TYPE ST_HW_OutputsEtherCAT_Bridge :
(**************************************************************************************
 * 	Application		:	BoxControl Framework
 *	Revision		:	$Revision: 355211 $
 *	Revision date	:	$Date: 2015-09-22 11:14:21 +0200 (Tue, 22 Sep 2015) $
 *	Last changed by	:	$Author: b7bolm $
 *	URL				:	$URL: http://almscdc.swisslog.com/repo/SWPD/Development/BoxControlFramework/20_Release/trunk/01_Software/BoxControlFramework/BoxControlFramework/JumpStart/11_Library/10_Application/11_Communication/12_MFCS/11_SIS/10_Base/FB_SIS_BaseDriver.TcPOU $
 *
 *	Purpose			:	Data for conveyor Subsystem interface over EtherCAT
 *
 * ------------------------------------------------------------------------------------
 *	Copyright Swisslog [IP AG], Switzerland. All rights reserved.
 * 
 * ------------------------------------------------------------------------------------
 *	
 * 	Revision History: 
 *
 * 	VERSION			DATE			INITIALS			DESCRIPTION
 *	0.1				01.01.2001		swl					Example
 *
 **************************************************************************************)
STRUCT
	STI					: ARRAY[1..20] OF ST_HW_InOutputsSTI_EtherCAT_Conveyor; // STI interface
END_STRUCT
END_TYPE

(* stored: Version 1.1.0.1, ProductVersion 3.1.4022.12
   DUT ST_HW_OutputsEtherCAT_Bridge: Id {5b57ca19-2371-4fbf-8cbf-2483a4247636} *)
